Universal Robots PolyScope program: WIE.urp

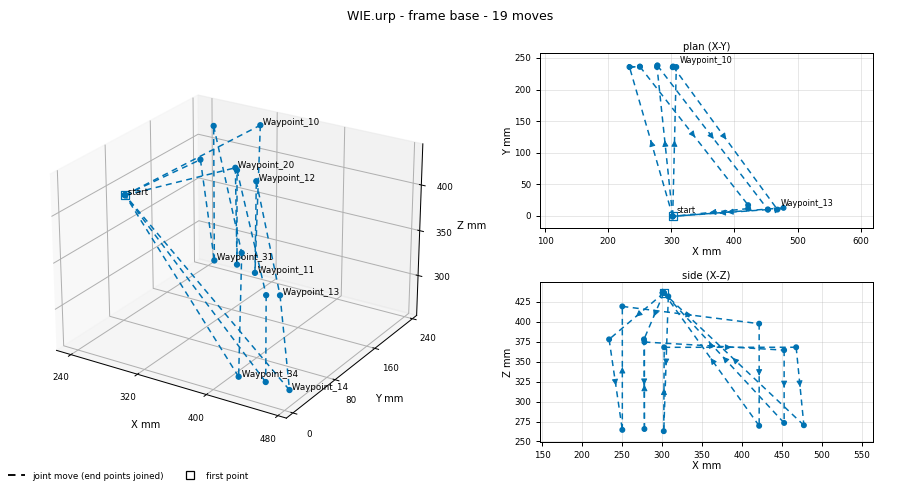
[picture p0: tool path of WIE.urp in frame base, 19 of 19 moves have a stored position in this frame; points joined in program order, loops and branches not executed]
Program WIE (installation=default directory=/programs/Students createdIn=5.11.9.1010452 lastSavedIn=5.11.9.1010452 robotSerialNumber=20225200364)
Calibrated DH parameters: a=[0.00002, -0.569483, -0.54992, -0.00001, -0.000036, 0]; d=[0.180894, -146.691669, 192.918669, -46.053088, 0.119778, 0.115602]; alpha=[1.571425, -0.001534, 0.003359, 1.568739, -1.571477, 0]; deltaTheta=[0, 0.376258, -0.101074, -0.275185, -0.000002, 0]
Robot Program (runOnlyOnce=false)
  MoveJ speed 60 deg/s, acceleration 80 deg/s^2 (useActiveTCP=true) feature=Base
    Waypoint start: TCP in base x=302.216 y=-0.86 z=436.116 mm, rx=2.2255 ry=-2.21 rz=0.004 rad; joints [35.142, -74.842, -127.962, -247.503, -90.011, -145.046] deg
    Waypoint Waypoint_10: TCP in base x=307.91 y=235.718 z=431.867 mm, rx=2.2254 ry=-2.2099 rz=0.0041 rad; joints [64.143, -85.346, -120.054, -244.975, -90.151, -116.03] deg
    Waypoint Waypoint_11: TCP in base x=302.204 y=235.296 z=262.887 mm, rx=2.2254 ry=-2.2099 rz=0.004 rad; joints [64.998, -96.131, -130.076, -224.166, -90.119, -115.104] deg
    URCap RG Grip (OnRobot, OnRobot A/S) dataModel(rg-target-force=40.0, rg-target-width=0.075, Variable(key=on_return, variable(name=on_return)))
    Waypoint Waypoint_12: TCP in base x=302.738 y=236.54 z=367.998 mm, rx=2.2254 ry=-2.2099 rz=0.004 rad; joints [64.988, -88.392, -124.549, -237.435, -90.148, -115.157] deg
    Waypoint Waypoint_13: TCP in base x=468.091 y=9.895 z=368.06 mm, rx=2.2254 ry=-2.21 rz=0.0041 rad; joints [23.117, -96.738, -115.688, -237.836, -89.92, -157.023] deg
    Waypoint Waypoint_14: TCP in base x=477.765 y=12.593 z=270.308 mm, rx=2.2256 ry=-2.2099 rz=0.004 rad; joints [22.952, -103.91, -119.177, -227.173, -89.901, -157.158] deg
    URCap RG Grip (OnRobot, OnRobot A/S) dataModel(rg-target-force=40.0, rg-target-width=0.1)
    Waypoint start: TCP in base x=302.216 y=-0.86 z=436.116 mm, rx=2.2255 ry=-2.21 rz=0.004 rad; joints [35.142, -74.842, -127.962, -247.503, -90.011, -145.046] deg
    Waypoint Waypoint_20: TCP in base x=277.405 y=235.742 z=377.988 mm, rx=2.2254 ry=-2.21 rz=0.0041 rad; joints [68.966, -85.577, -125.993, -238.804, -90.172, -111.183] deg
    Waypoint Waypoint_21: TCP in base x=277.944 y=238.04 z=265.65 mm, rx=2.2255 ry=-2.2098 rz=0.0041 rad; joints [69.043, -94.232, -131.843, -224.302, -90.143, -111.064] deg
    URCap RG Grip (OnRobot, OnRobot A/S) dataModel(rg-target-force=40.0, rg-target-width=0.075, Variable(key=on_return, variable=on_return))
    Waypoint Waypoint_22: TCP in base x=277.969 y=238.05 z=374.593 mm, rx=2.2255 ry=-2.21 rz=0.0042 rad; joints [69.022, -85.999, -126.011, -238.365, -90.169, -111.129] deg
    Waypoint Waypoint_23: TCP in base x=453.012 y=9.898 z=364.466 mm, rx=2.2254 ry=-2.2101 rz=0.0041 rad; joints [23.928, -95.507, -117.516, -237.242, -89.923, -156.208] deg
    Waypoint Waypoint_24: TCP in base x=453.022 y=9.9 z=273.227 mm, rx=2.2253 ry=-2.2101 rz=0.0041 rad; joints [23.937, -101.577, -121.868, -226.819, -89.903, -156.162] deg
    URCap RG Grip (OnRobot, OnRobot A/S) dataModel(rg-target-force=40.0, rg-target-width=0.1)
    Waypoint start: TCP in base x=302.216 y=-0.86 z=436.116 mm, rx=2.2255 ry=-2.21 rz=0.004 rad; joints [35.142, -74.842, -127.962, -247.503, -90.011, -145.046] deg
    Waypoint Waypoint_30: TCP in base x=233.725 y=235.747 z=377.969 mm, rx=2.2254 ry=-2.2099 rz=0.0041 rad; joints [76.908, -81.844, -129.218, -239.315, -90.225, -103.25] deg
    Waypoint Waypoint_31: TCP in base x=250.276 y=236.27 z=264.563 mm, rx=2.2254 ry=-2.2099 rz=0.0041 rad; joints [73.795, -92.122, -134.293, -223.965, -90.174, -106.308] deg
    URCap RG Grip (OnRobot, OnRobot A/S) dataModel(rg-target-force=40.0, rg-target-width=0.075, Variable(key=on_return, variable=on_return))
    Waypoint Waypoint_32: TCP in base x=250.27 y=236.251 z=419.264 mm, rx=2.2253 ry=-2.2098 rz=0.0042 rad; joints [73.762, -80.998, -125.195, -244.193, -90.212, -106.412] deg
    Waypoint Waypoint_33: TCP in base x=421.722 y=16.909 z=397.603 mm, rx=2.2254 ry=-2.2098 rz=0.0041 rad; joints [26.745, -90.618, -118.854, -240.815, -89.941, -153.412] deg
    Waypoint Waypoint_34: TCP in base x=421.735 y=11.412 z=269.635 mm, rx=2.2254 ry=-2.2099 rz=0.0042 rad; joints [26.027, -99.105, -125.508, -225.666, -89.906, -154.075] deg
    URCap RG Grip (OnRobot, OnRobot A/S) dataModel(rg-target-force=40.0, rg-target-width=0.1)
    Waypoint start: TCP in base x=302.216 y=-0.86 z=436.116 mm, rx=2.2255 ry=-2.21 rz=0.004 rad; joints [35.142, -74.842, -127.962, -247.503, -90.011, -145.046] deg
    Halt
